INTERFACE I_MotionAxisMoveAbsolute

END_INTERFACE

(* stored: Version 1.1.0.1
   Itf I_MotionAxisMoveAbsolute: Id {943c1688-37bf-4c0b-8ef2-246b1c0d27a0} *)
